FUNCTION_BLOCK FB_MachineModeFromEPICS
(*
Readback options are:

0 – NC (normal conducting, copper linac)

1 – SC (superconducting linac)

2 – Misconfigured (something in link node not set correctly.

*)
VAR_IN_OUT
    BP : ST_BeamParams;
    fbMPS_MachineMode : FB_LREALFromEPICS;
    FFO : FB_HardwareFFOutput;
END_VAR
VAR_OUTPUT
    xError : BOOL;
END_VAR
VAR

    ffModeReadBack : FB_FastFault := (
        i_DevName := 'Arbiter',
        i_Desc := 'Issue with Machine mode readback from Accelerator. Gateway or EPICS connection. Must be fixed.',
        i_TypeCode := 16#313,
        i_xAutoReset:=True);
END_VAR
VAR CONSTANT
    cFailSafeMM : USINT := 3;
END_VAR

fbMPS_MachineMode();

IF fbMPS_MachineMode.bValid THEN
    BP.nMachineMode := LREAL_TO_USINT(fbMPS_MachineMode.fValue);
ELSE
    BP.nMachineMode := cFailSafeMM;
END_IF

ffModeReadBack(i_xOK:=(fbMPS_MachineMode.bValid) AND fbMPS_MachineMode.fValue <2 , io_fbFFHWO:=FFO);

BP.xValid R= NOT fbMPS_MachineMode.bValid;

END_FUNCTION_BLOCK

(* stored: Version 1.1.0.1, ProductVersion 3.1.4022.18
   POU FB_MachineModeFromEPICS: Id {e77c5ce7-1295-45e2-913d-511a3f59fc41}, SpecialFunc None *)
